KUKA KRL program: MasRef_User.src, MasRef_User.dat

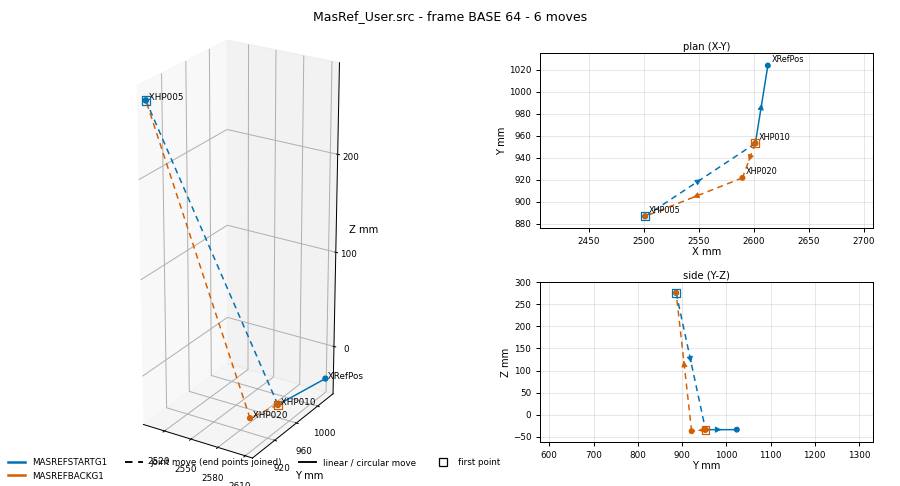
[picture p0: tool path of MasRef_User.src in frame BASE 64, 6 of 8 moves have a stored position in this frame; points joined in program order, loops and branches not executed]
--- MasRef_User.src ---
&ACCESS RVP4
&REL 16
&COMMENT MasRef User
&PARAM TEMPLATE = C:\KRC\roboter\template\vg_appl
&PARAM DISKPATH = KRC:\R1\Program
DEF MasRef_User( )
;FOLD ; Anlagenbezeichn: HC53_C    Stations-Nr: 060RB_100;%{PE}
;FOLD Parameters ;%{h}
;Params IlfProvider=kukaroboter.basistech.inlineforms.comments.comment; Kuka.Content=Anlagenbezeichn: HC53_C    Stations-Nr: 060RB_100
;ENDFOLD
;ENDFOLD
;FOLD ; Stand / Version: V1.0;%{PE}
;FOLD Parameters ;%{h}
;Params IlfProvider=kukaroboter.basistech.inlineforms.comments.comment; Kuka.Content=Stand / Version: V1.0
;ENDFOLD
;ENDFOLD
;FOLD ; Name Bearbeiter: EBZ-AE;%{PE}
;FOLD Parameters ;%{h}
;Params IlfProvider=kukaroboter.basistech.inlineforms.comments.comment; Kuka.Content=Name Bearbeiter: EBZ-AE
;ENDFOLD
;ENDFOLD
;FOLD ; Translator Version:29.01.2024 - Version 15.08;%{PE}
;FOLD Parameters ;%{h}
;Params IlfProvider=kukaroboter.basistech.inlineforms.comments.comment; Kuka.Content=Translator Version:29.01.2024 - Version 15.08
;ENDFOLD
;ENDFOLD
END

GLOBAL DEF MASREFSTARTG1()
;FOLD INI;%{PE}
  ;FOLD BASISTECH INI
    GLOBAL INTERRUPT DECL 3 WHEN $STOPMESS==TRUE DO IR_STOPM ( )
    INTERRUPT ON 3
    BAS (#INITMOV,0 )
  ;ENDFOLD (BASISTECH INI)
  ;FOLD USER INI
    ;Make your modifications here
  ;ENDFOLD (USER INI)
;ENDFOLD (INI)
;FOLD Teach path and position for reference group 1
;ENDFOLD

;Collision detection - Process Motion 30
;FOLD COLLDETECT UseDataSet DataSet[30];%{PE}%R 8.5.19,%MKUKATPBASIS,%CTQ_MON,%VTQ_CDSET,%P 2:TQ_CDSET, 4:30
USE_CD_PARAMS(30)
;ENDFOLD


;FOLD ; This program has been cleaned by KANERT_Makro. High risk of crash!!! Check the program carefully before deleting this comment. ;%{PE}
;FOLD Parameters ;%{h}
;Params IlfProvider=kukaroboter.basistech.inlineforms.comments.comment; Kuka.Content=This program has been cleaned by KANERT_Makro. High risk of crash!!! Check the program carefully before deleting this comment.
;ENDFOLD
WAIT FOR FALSE
;ENDFOLD
WAIT FOR FALSE ;STATUS
;PROGRAM CHECKED BY: p.kanert
;COLLISIONS NOT CHECKED

WAIT FOR nearE6Axis (XHOME)
;FOLD PTP HOME Vel=100 % DEFAULT;%{PE}
;FOLD Parameters ;%{h}
;Params IlfProvider=kukaroboter.basistech.inlineforms.movement.old; Kuka.IsGlobalPoint=False; Kuka.PointName=HOME; Kuka.BlendingEnabled=False; Kuka.MoveDataPtpName=DEFAULT; Kuka.VelocityPtp=100; Kuka.CurrentCDSetIndex=0; Kuka.MovementParameterFieldEnabled=True; IlfCommand=PTP
;ENDFOLD
$BWDSTART = FALSE
PDAT_ACT = PDEFAULT
FDAT_ACT = FHOME
BAS(#PTP_PARAMS, 100.0)
SET_CD_PARAMS (0)
PTP XHOME
;ENDFOLD

;Dynamische Pruefung Teil vorhanden
;FOLD PartPresent.CheckOff #1: 5277, #2: 5278, #3: 1025, #4: 1025, #5: 1025, #6: 1025, Bounce Time: 100, Constant: Yes ;%{PE}
CheckPartPresent(5277,5278,1025,1025,1025,1025,100, True,FALSE)
;ENDFOLD

;Greifer-Ventile betatigen/pruefen
;FOLD DAI_GripValveCheck.Valve2 State:Fixierstift Ausfahren Gs, 060GRH101-QM1;%{PE}%
CheckValveState(2,1)
;ENDFOLD
;FOLD DAI_GripValveCheck.Valve3 State:Spanner Oeffnen Gs, 060GRH101-QM2;%{PE}%
CheckValveState(3,1)
;ENDFOLD
;FOLD DAI_GripValveCheck.Valve4 State:Spanner Oeffnen Gs, 060GRH101-QM3;%{PE}%
CheckValveState(4,1)
;ENDFOLD

;Collision detection - Process Motion 27
;FOLD COLLDETECT UseDataSet DataSet[27];%{PE}%R 8.5.19,%MKUKATPBASIS,%CTQ_MON,%VTQ_CDSET,%P 2:TQ_CDSET, 4:27
USE_CD_PARAMS(27)
;ENDFOLD

;FOLD PTP HP005 CONT Vel=100 % PDAT1 Tool[62]:Safe-Ref Base[64]:Zero;%{PE}
;FOLD Parameters ;%{h}
;Params IlfProvider=kukaroboter.basistech.inlineforms.movement.old; Kuka.IsGlobalPoint=False; Kuka.PointName=HP005; Kuka.BlendingEnabled=True; Kuka.MoveDataPtpName=PDAT1; Kuka.VelocityPtp=100; Kuka.CurrentCDSetIndex=0; Kuka.MovementParameterFieldEnabled=True; IlfCommand=PTP
;ENDFOLD
$BWDSTART = FALSE
PDAT_ACT = PPDAT1
FDAT_ACT = FHP005
BAS(#PTP_PARAMS, 100.0)
SET_CD_PARAMS (0)
PTP XHP005 C_Dis
;ENDFOLD
;FOLD PTP HP010 Vel=100 % PDAT2 Tool[62]:Safe-Ref Base[64]:Zero ;%{PE}
;FOLD Parameters ;%{h}
;Params IlfProvider=kukaroboter.basistech.inlineforms.movement.old; Kuka.IsGlobalPoint=False; Kuka.PointName=HP010; Kuka.BlendingEnabled=False; Kuka.MoveDataPtpName=PDAT2; Kuka.VelocityPtp=100; Kuka.CurrentCDSetIndex=0; Kuka.MovementParameterFieldEnabled=True; IlfCommand=PTP
;ENDFOLD
$BWDSTART = FALSE
PDAT_ACT = PPDAT2
FDAT_ACT = FHP010
BAS(#PTP_PARAMS, 100.0)
SET_CD_PARAMS (0)
PTP XHP010
;ENDFOLD
;FOLD LIN RefPos Vel=0.5 m/s CPDAT3 Tool[62]:Safe-Ref Base[64]:Zero ;%{PE}
;FOLD Parameters ;%{h}
;Params IlfProvider=kukaroboter.basistech.inlineforms.movement.old; Kuka.IsGlobalPoint=False; Kuka.PointName=RefPos; Kuka.BlendingEnabled=False; Kuka.MoveDataName=CPDAT3; Kuka.VelocityPath=0.5; Kuka.CurrentCDSetIndex=0; Kuka.MovementParameterFieldEnabled=True; IlfCommand=LIN
;ENDFOLD
$BWDSTART = FALSE
LDAT_ACT = LCPDAT3
FDAT_ACT = FRefPos
BAS(#CP_PARAMS, 0.5)
SET_CD_PARAMS (0)
LIN XRefPos
;ENDFOLD

END

GLOBAL DEF MASREFBACKG1()
;FOLD Teach path back for reference group 1
;ENDFOLD

;Collision detection - Process Motion 27
;FOLD COLLDETECT UseDataSet DataSet[27];%{PE}%R 8.5.19,%MKUKATPBASIS,%CTQ_MON,%VTQ_CDSET,%P 2:TQ_CDSET, 4:27
USE_CD_PARAMS(27)
;ENDFOLD

;FOLD LIN HP015 Vel=0.5 m/s CPDAT4 Tool[62]:Safe-Ref Base[64]:Zero ;%{PE}
;FOLD Parameters ;%{h}
;Params IlfProvider=kukaroboter.basistech.inlineforms.movement.old; Kuka.IsGlobalPoint=False; Kuka.PointName=HP015; Kuka.BlendingEnabled=False; Kuka.MoveDataName=CPDAT4; Kuka.VelocityPath=0.5; Kuka.CurrentCDSetIndex=0; Kuka.MovementParameterFieldEnabled=True; IlfCommand=LIN
;ENDFOLD
$BWDSTART = FALSE
LDAT_ACT = LCPDAT4
FDAT_ACT = FHP015
BAS(#CP_PARAMS, 0.5)
SET_CD_PARAMS (0)
LIN XHP015
;ENDFOLD
;FOLD PTP HP020 Vel=100 % PDAT5 Tool[62]:Safe-Ref Base[64]:Zero ;%{PE}
;FOLD Parameters ;%{h}
;Params IlfProvider=kukaroboter.basistech.inlineforms.movement.old; Kuka.IsGlobalPoint=False; Kuka.PointName=HP020; Kuka.BlendingEnabled=False; Kuka.MoveDataPtpName=PDAT5; Kuka.VelocityPtp=100; Kuka.CurrentCDSetIndex=0; Kuka.MovementParameterFieldEnabled=True; IlfCommand=PTP
;ENDFOLD
$BWDSTART = FALSE
PDAT_ACT = PPDAT5
FDAT_ACT = FHP020
BAS(#PTP_PARAMS, 100.0)
SET_CD_PARAMS (0)
PTP XHP020
;ENDFOLD
;FOLD PTP HP025 CONT Vel=100 % PDAT6 Tool[62]:Safe-Ref Base[64]:Zero ;%{PE}
;FOLD Parameters ;%{h}
;Params IlfProvider=kukaroboter.basistech.inlineforms.movement.old; Kuka.IsGlobalPoint=False; Kuka.PointName=HP025; Kuka.BlendingEnabled=True; Kuka.MoveDataPtpName=PDAT6; Kuka.VelocityPtp=100; Kuka.CurrentCDSetIndex=0; Kuka.MovementParameterFieldEnabled=True; IlfCommand=PTP
;ENDFOLD
$BWDSTART = FALSE
PDAT_ACT = PPDAT6
FDAT_ACT = FHP025
BAS(#PTP_PARAMS, 100.0)
SET_CD_PARAMS (0)
PTP XHP025 C_Dis
;ENDFOLD

;Collision detection - Global/HOME/Guebergabe
;FOLD COLLDETECT UseDataSet DataSet[30];%{PE}%R 8.5.19,%MKUKATPBASIS,%CTQ_MON,%VTQ_CDSET,%P 2:TQ_CDSET, 4:30
USE_CD_PARAMS( 30)
;ENDFOLD

;FOLD PTP HOME Vel=100 % DEFAULT;%{PE}
;FOLD Parameters ;%{h}
;Params IlfProvider=kukaroboter.basistech.inlineforms.movement.old; Kuka.IsGlobalPoint=False; Kuka.PointName=HOME; Kuka.BlendingEnabled=False; Kuka.MoveDataPtpName=DEFAULT; Kuka.VelocityPtp=100; Kuka.CurrentCDSetIndex=0; Kuka.MovementParameterFieldEnabled=True; IlfCommand=PTP
;ENDFOLD
$BWDSTART = FALSE
PDAT_ACT = PDEFAULT
FDAT_ACT = FHOME
BAS(#PTP_PARAMS, 100.0)
SET_CD_PARAMS (0)
PTP XHOME
;ENDFOLD

;Collision detection - Off
;FOLD COLLDETECT Off ;%{PE}
 ;FOLD Parameters ;%{h}
 ;Params IlfProvider=kukaroboter.basistech.inlineforms.colldetect.off; CollDetect.Command=Off
 ;ENDFOLD
 USE_CD_PARAMS(0)
 ;ENDFOLD

END

GLOBAL DEF MASREFSTARTG2()
;FOLD Teach path and position for reference group 2
;ENDFOLD

END

GLOBAL DEF MASREFBACKG2()
;FOLD Teach path back for reference group 2
;ENDFOLD

END

GLOBAL DEF MASREFSTARTG3()
;FOLD Teach path and position for reference group 3
;ENDFOLD

END

GLOBAL DEF MASREFBACKG3()
;FOLD Teach path back for reference group 3
;ENDFOLD
END

--- MasRef_User.dat ---
&ACCESS  RVP
&COMMENT MasRef User
&PARAM DISKPATH = KRC:\R1\Program
&PARAM TEMPLATE = C:\KRC\roboter\template\vg_appl
&REL 1
DEFDAT  MASREF_USER PUBLIC
;FOLD EXTERNAL DECLARATIONS;%{PE}%MKUKATPBASIS,%CEXT,%VCOMMON,%P
;FOLD BASISTECH EXT;%{PE}%MKUKATPBASIS,%CEXT,%VEXT,%P
EXT  BAS (BAS_COMMAND  :IN,REAL  :IN )
DECL INT SUCCESS
;ENDFOLD (BASISTECH EXT)
;FOLD USER EXT;%{E}%MKUKATPUSER,%CEXT,%VEXT,%P
;Make your modifications here
;ENDFOLD (USER EXT)
;FOLD COLLISION
EXT  COLLSTOP (INT  :IN,INT  :IN )
;ENDFOLD  (Collision)
;ENDFOLD (EXTERNAL DECLERATIONS)
;FOLD reference groups
DECL GLOBAL CONST INT MASREFg_GroupSequence[3] ; contains reference groups to test
MASREFg_GroupSequence[1]=1
MASREFg_GroupSequence[2]=0
MASREFg_GroupSequence[3]=0
;ENDFOLD (reference groups)
DECL BASIS_SUGG_T LAST_BASIS={POINT1[] "P0                      ",POINT2[] "P0                      ",CP_PARAMS[] "CPDAT0                  ",PTP_PARAMS[] "PDAT0                   ",CONT[] "                        ",CP_VEL[] "2.0                     ",PTP_VEL[] "100                     ",SYNC_PARAMS[] "SYNCDAT                 ",SPL_NAME[] "S0                      ",A_PARAMS[] "ADAT0                   "}
DECL MODULEPARAM_T LAST_TP_PARAMS={PARAMS[] "Kuka.PointName=HP025; Kuka.FrameData.base_no=64; Kuka.FrameData.tool_no=62; Kuka.FrameData.ipo_frame=#BASE; Kuka.FrameData.point2=; Kuka.isglobalpoint=False; Kuka.MoveDataPtpName=PDAT5; Kuka.MovementDataPdat.apo_mode=#CDIS; Kuka.MovementDataPdat.apo_dist=1000; Kuka.MovementData.vel=0.5; Kuka.MovementData.acc=100; Kuka.MovementData.exax_ign=0; Kuka.VelocityPtp=100; Kuka.BlendingEnabled=False; Kuka.APXEnabled=False; Kuka.CurrentCDSetIndex=0; Kuka.MoveDataName=CPDAT7; Kuka.MovementData.cb={AUX_PT {ORI #CONSIDER,E1 #CONSIDER,E2 #CONSIDER,E3 #CONSIDER,E4 #CONSIDER,E5 #CONSIDER,E6 #CONSIDER},TARGET_PT {ORI #INTERPOLATE,E1 #INTERPOLATE,E2 #INTERPOLATE,E3 #INTERPOLATE,E4 #INTERPOLATE,E5 #INTERPOLATE,E6 #INTERPOLATE}}; Kuka.MovementData.apo_fac=50; Kuka.MovementData.apo_dist=100; Kuka.MovementData.axis_acc=100; Kuka.MovementData.axis_vel=100; Kuka.MovementData.circ_typ=#BASE; Kuka.MovementData.jerk_fac=50; Kuka.MovementData.ori_typ=#VAR; Kuka.VelocityPath=0.5; PARTPRESENT.NUMPPOFF1=5277; PARTPRESENT.NUMPPOFF2=5278; PARTPRESENT.NUMPPOFF3=1025; PARTPRESENT.NUMPPOFF4=1025; PARTPRESENT.NUMPPOFF5=1025; PARTPRESENT.NUMPPOFF6=1025; PARTPRESENT.NUMBOUNCE=100; PARTPRESENT.LSTBOUNCEENABLED=True; PARTPRESENT.NUMPP1=51; PARTPRESENT.NUMPP2=0; PARTPRESENT.NUMPP3=0; PARTPRESENT.NUMPP4=0; PARTPRESENT.NUMPP5=0; PARTPRESENT.NUMPP6=0"}

; E6POS Declarations
DECL E6POS XHP005={X 2501.09668,Y 886.753540,Z 275.450867,A -10.0038977,B 179.148163,C -0.523956478,S 18,T 3,E1 100.000,E2 0.0,E3 0.0,E4 0.0,E5 0.0,E6 0.0}
DECL E6POS XHP010={X 2601.28369,Y 953.137146,Z -33.6053314,A 169.995911,B 0.0187745374,C -179.983780,S 18,T 3,E1 100.000,E2 0.0,E3 0.0,E4 0.0,E5 0.0,E6 0.0}
DECL E6POS XRefPos={X 2612.66260,Y 1023.90460,Z -33.5625648,A 170.000092,B -0.000144479185,C -179.999695,S 18,T 3,E1 100.000,E2 0.0,E3 0.0,E4 0.0,E5 0.0,E6 0.0}
DECL E6POS XHP015={X 2601.28076,Y 953.134094,Z -33.6063881,A 169.995956,B 0.0187369511,C -179.983749,S 18,T 3,E1 100.000,E2 0.0,E3 0.0,E4 0.0,E5 0.0,E6 0.0}
DECL E6POS XHP020={X 2589.54199,Y 921.756,Z -37.0501785,A -10.0000019,B 179.999954,C 0.0,S 18,T 3,E1 100.000,E2 0.0,E3 0.0,E4 0.0,E5 0.0,E6 0.0}
DECL E6POS XHP025={X 2501.09668,Y 886.753540,Z 275.450867,A -10.0038977,B 179.148163,C -0.523956478,S 18,T 3,E1 100.000,E2 0.0,E3 0.0,E4 0.0,E5 0.0,E6 0.0}

; PDAT/LDAT Declarations
DECL PDAT PPDAT1={VEL 100.000,ACC 100.000,APO_DIST 1000.00,APO_MODE #CDIS,GEAR_JERK 50.0000,EXAX_IGN 0}
DECL PDAT PPDAT2={VEL 100.000,ACC 100.000,APO_DIST 1000.00,APO_MODE #CDIS,GEAR_JERK 50.0000,EXAX_IGN 0}
DECL LDAT LCPDAT3={VEL 0.500000,ACC 100.000,APO_DIST 0.0,APO_FAC 50.0000,AXIS_VEL 100.000,AXIS_ACC 100.000,ORI_TYP #VAR,CIRC_TYP #BASE,JERK_FAC 50.0000,GEAR_JERK 50.0000,EXAX_IGN 0}
DECL LDAT LCPDAT4={VEL 0.500000,ACC 100.000,APO_DIST 100.000,APO_FAC 50.0000,AXIS_VEL 100.000,AXIS_ACC 100.000,ORI_TYP #VAR,CIRC_TYP #BASE,JERK_FAC 50.0000,GEAR_JERK 50.0000,EXAX_IGN 0,CB {AUX_PT {ORI #CONSIDER,E1 #CONSIDER,E2 #CONSIDER,E3 #CONSIDER,E4 #CONSIDER,E5 #CONSIDER,E6 #CONSIDER},TARGET_PT {ORI #INTERPOLATE,E1 #INTERPOLATE,E2 #INTERPOLATE,E3 #INTERPOLATE,E4 #INTERPOLATE,E5 #INTERPOLATE,E6 #INTERPOLATE}}}
DECL PDAT PPDAT5={VEL 100.000,ACC 100.000,APO_DIST 500.000,APO_MODE #CDIS,GEAR_JERK 100.000,EXAX_IGN 0}
DECL PDAT PPDAT6={VEL 100.000,ACC 100.000,APO_DIST 1000.00,APO_MODE #CDIS,GEAR_JERK 50.0000,EXAX_IGN 0}

; FDAT Declarations
DECL FDAT FHOME={TOOL_NO 62,BASE_NO 64,IPO_FRAME #BASE,POINT2[] " "}
DECL FDAT FHP005={TOOL_NO 62,BASE_NO 64,IPO_FRAME #BASE,POINT2[] " "}
DECL FDAT FHP010={TOOL_NO 62,BASE_NO 64,IPO_FRAME #BASE,POINT2[] " "}
DECL FDAT FRefPos={TOOL_NO 62,BASE_NO 64,IPO_FRAME #BASE,POINT2[] " "}
DECL FDAT FHP015={TOOL_NO 62,BASE_NO 64,IPO_FRAME #BASE,POINT2[] " "}
DECL FDAT FHP020={TOOL_NO 62,BASE_NO 64,IPO_FRAME #BASE,POINT2[] " "}
DECL FDAT FHP025={TOOL_NO 62,BASE_NO 64,IPO_FRAME #BASE,POINT2[] " "}

ENDDAT
